// TIA Portal V17 export
// export: Created 2022-07-20T07:01:33.0729322Z, ExportSetting WithDefaults, DisplayName Totally Integrated Automation Portal, DisplayVersion V17, DisplayName TIA Portal Openness, DisplayVersion V17, DisplayName TIA Portal Version Control Interface, DisplayVersion V17, DisplayName SINAMICS Startdrive Advanced, DisplayVersion V17, DisplayName SINAMICS Startdrive G130, G150, S120, S150, SINAMICS MV, S210, DisplayVersion V17, DisplayName SINAMICS Startdrive G110M, G120, G120C, G120D, G120P, G115D, DisplayVersion V17, DisplayName STEP 7 Professional, DisplayVersion V17, DisplayName STEP 7 Safety, DisplayVersion V17, DisplayName WinCC Advanced, DisplayVersion V17
FUNCTION_BLOCK "FB10310_DegassingPlant"   // FB10310, LAD
{ S7_Optimized_Access := 'TRUE' }
VERSION : 0.1
// stored: AutoNumber false, IsIECCheckEnabled false, IsRetainMemResEnabled false, MemoryReserve 100, SetENOAutomatically false, UDAEnableTagReadback false
   VAR_INPUT
      Acknwoledge : Bool;
      PressureSensorRawValue : Int;
      DegassingSystemSetPoint : Real;
   END_VAR
   VAR_OUTPUT
      ActiveDegassingPump : Bool;
      ActiveDegassingSolenoidValve : Bool;
      DegassingSystemRegulationInProgress : Bool;
      DegassingSystemInError : Bool;
      DegassingSystemActualPressure : Real;
   END_VAR
   VAR_IN_OUT
      RequestActiveDegassingSystemAutoregulation : Bool;
      RequestStopDegassingSystemAutoregulation : Bool;
   END_VAR
   VAR
      DegassingSystemAutoregulationStateDiagram : Int;
      CalibrationDataX_1 : Real := 0.0;
      CalibrationDataX_2 : Real := 27648.0;
      CalibrationDataY_1 : Real := 0.0;
      CalibrationDataY_2 : Real := -950.0;
      R_TRIG_RequestActiveDegassingSystemAutoregulation { S7_SetPoint := 'True'} : R_TRIG;
      R_TRIG_RequestStopDegassingSystemAutoregulation { S7_SetPoint := 'True'} : R_TRIG;
      TON_ActiveDegassingPump { S7_SetPoint := 'True'} : TON_TIME;
      TON_DegassingSystemTimeout { S7_SetPoint := 'True'} : TON_TIME;
      FB10030_AnalogicalSensor_DegassingPressureSensor { S7_SetPoint := 'True'} : "FB10030_AnalogicalSensor";
   END_VAR
   VAR CONSTANT
      WAIT_FOR_DEGASSING_SYSTEM_AUTOREGULATION_REQUEST : Int := 0;
      DEGASSING_SYSTEM_PRESSURE_UNDER_SETPOINT : Int := 10;
      DEGASSING_SYSTEM_PRESSURE_OVER_SETPOINT : Int := 20;
      DEGASSING_SYSTEM_AUTOREGULATION_REQUEST_DONE : Int := 30;
   END_VAR
BEGIN

REGION Network 1 (SCL): First Scan
   IF "FirstScan" THEN
       #DegassingSystemAutoregulationStateDiagram := #WAIT_FOR_DEGASSING_SYSTEM_AUTOREGULATION_REQUEST;
   END_IF;
END_REGION

REGION Network 2 (SCL): Edge Signals & Timers
   REGION EDGE SIGNALS
       #R_TRIG_RequestActiveDegassingSystemAutoregulation(CLK := #RequestActiveDegassingSystemAutoregulation);
       #R_TRIG_RequestStopDegassingSystemAutoregulation(CLK := #RequestStopDegassingSystemAutoregulation);
   END_REGION

   REGION TIMERS
       #TON_ActiveDegassingPump(IN := #ActiveDegassingPump,
                                PT := T#40s);
       #TON_DegassingSystemTimeout(IN := #ActiveDegassingPump,
                                   PT := T#2m);
   END_REGION
END_REGION

REGION Network 3: Degassing Pressure Sensor Management
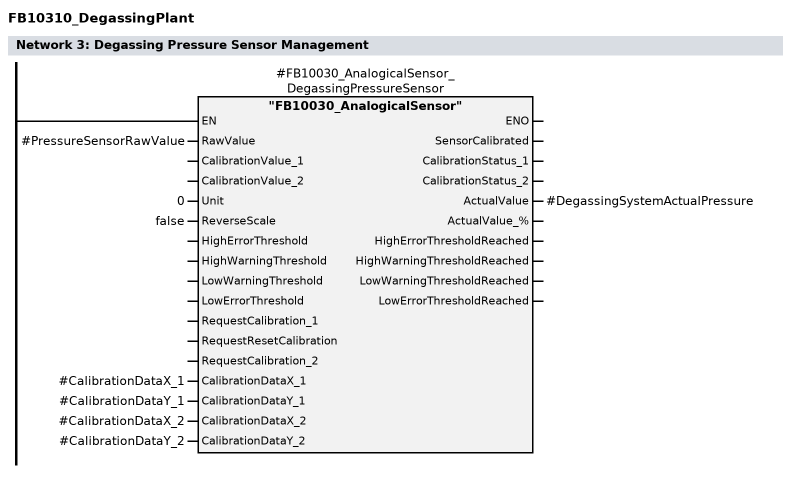
   RUNG wire#powerrail
      #FB10030_AnalogicalSensor_DegassingPressureSensor(RawValue := #PressureSensorRawValue, CalibrationValue_1 :=, CalibrationValue_2 :=, Unit := 0, ReverseScale := false, HighErrorThreshold :=, HighWarningThreshold :=, LowWarningThreshold :=, LowErrorThreshold :=, RequestCalibration_1 :=, RequestResetCalibration :=, RequestCalibration_2 :=, CalibrationDataX_1 := #CalibrationDataX_1, CalibrationDataY_1 := #CalibrationDataY_1, CalibrationDataX_2 := #CalibrationDataX_2, CalibrationDataY_2 := #CalibrationDataY_2, SensorCalibrated =>, CalibrationStatus_1 =>, CalibrationStatus_2 =>, ActualValue => #DegassingSystemActualPressure, "ActualValue_%" =>, HighErrorThresholdReached =>, HighWarningThresholdReached =>, LowWarningThresholdReached =>, LowErrorThresholdReached =>)
   END_RUNG
   // the same network as SCL:
   #FB10030_AnalogicalSensor_DegassingPressureSensor(RawValue := #PressureSensorRawValue,   // "FB10030_AnalogicalSensor"
                           Unit := 0,
                           ReverseScale := false,
                           CalibrationDataX_1 := #CalibrationDataX_1,
                           CalibrationDataY_1 := #CalibrationDataY_1,
                           CalibrationDataX_2 := #CalibrationDataX_2,
                           CalibrationDataY_2 := #CalibrationDataY_2,
                           ActualValue => #DegassingSystemActualPressure);
END_REGION

REGION Network 4 (SCL): Degassing System Management
   CASE #DegassingSystemAutoregulationStateDiagram OF
       #WAIT_FOR_DEGASSING_SYSTEM_AUTOREGULATION_REQUEST:
           IF #R_TRIG_RequestActiveDegassingSystemAutoregulation.Q THEN
               #DegassingSystemRegulationInProgress := TRUE;
               #DegassingSystemAutoregulationStateDiagram := #DEGASSING_SYSTEM_PRESSURE_UNDER_SETPOINT;
           END_IF;
       #DEGASSING_SYSTEM_PRESSURE_UNDER_SETPOINT:
           IF #DegassingSystemActualPressure > (#DegassingSystemSetPoint - (#DegassingSystemSetPoint/100.0)) THEN
               #ActiveDegassingPump := TRUE;
               #ActiveDegassingSolenoidValve := FALSE;
           ELSIF #DegassingSystemActualPressure <= #DegassingSystemSetPoint THEN
               #ActiveDegassingPump := FALSE;
               #ActiveDegassingSolenoidValve := TRUE;
           END_IF;
       #DEGASSING_SYSTEM_AUTOREGULATION_REQUEST_DONE:
           #ActiveDegassingPump := FALSE;
           #ActiveDegassingSolenoidValve := TRUE;
           #DegassingSystemRegulationInProgress := FALSE;
           #DegassingSystemAutoregulationStateDiagram := #WAIT_FOR_DEGASSING_SYSTEM_AUTOREGULATION_REQUEST;
   END_CASE;

   IF #R_TRIG_RequestStopDegassingSystemAutoregulation.Q THEN
       #DegassingSystemAutoregulationStateDiagram := #DEGASSING_SYSTEM_AUTOREGULATION_REQUEST_DONE;
   END_IF;
END_REGION

REGION Network 5 (SCL): Error Management
   REGION DEGASSING SYSTEM
       IF #TON_DegassingSystemTimeout.Q THEN
           #DegassingSystemAutoregulationStateDiagram := #DEGASSING_SYSTEM_AUTOREGULATION_REQUEST_DONE;
           #DegassingSystemInError := TRUE;
       END_IF;

       IF #Acknwoledge THEN
           #DegassingSystemInError := FALSE;
       END_IF;
   END_REGION
END_REGION
END_FUNCTION_BLOCK
